FUNCTION_BLOCK FB_Button_1
VAR_INPUT
	bButtonPress : BOOL;
END_VAR
VAR_OUTPUT
	nCounter: INT;
END_VAR
VAR
END_VAR

END_FUNCTION_BLOCK

(* stored: Version 1.1.0.1
   POU FB_Button_1: Id {8bc74369-b140-45ba-9250-a27cb5ef27e3}, SpecialFunc None *)
